SUBAPPLICATION SR_TO_QX_TRIG_EO (* SET/RESET-Latch (E_SR) auf QX, mit Event-Echo EO1 nach jeder steigenden Flanke des Latch-Zustands. Generisch. *)
  (* Standard: 61499-2 *)
  (* Version 1.0, 2026-09-09, Franz Höpfinger, Meisterschulen am Ostbahnhof, Ausgelagert aus Uebung_026_sub zur Wiederverwendung. *)
  PACKAGE MyLib::sys;
  IMPORT logiBUS::io::DQ::logiBUS_DO;
  IMPORT logiBUS::io::DQ::logiBUS_DO_S;
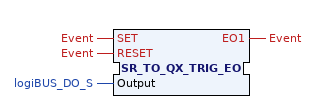
  EVENT_INPUT
    SET;
    RESET;
  END_EVENT
  EVENT_OUTPUT
    EO1;
  END_EVENT
  VAR_INPUT
    Output : logiBUS::io::DQ::logiBUS_DO_S := logiBUS_DO::Invalid; (* Identify the Output Output_Q1..Q8 *)
  END_VAR
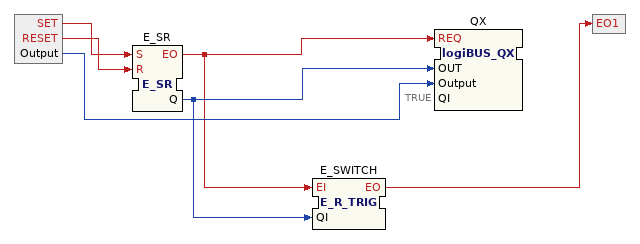
  FBS
    E_SR : iec61499::events::E_SR;
    QX : logiBUS::io::DQ::logiBUS_QX(QI := TRUE);
    E_SWITCH : iec61499::events::E_R_TRIG;
  END_FBS
  EVENT_CONNECTIONS
    E_SR.EO TO QX.REQ;
    E_SR.EO TO E_SWITCH.EI;
    SET TO E_SR.S;
    RESET TO E_SR.R;
    E_SWITCH.EO TO EO1;
  END_CONNECTIONS
  DATA_CONNECTIONS
    E_SR.Q TO QX.OUT;
    E_SR.Q TO E_SWITCH.QI;
    Output TO QX.Output;
  END_CONNECTIONS
END_SUBAPPLICATION
